// Mitsubishi GX Works2 project: tutor09_webmonitor   PLC: FX1N/FX1NC

PROGRAM MAIN
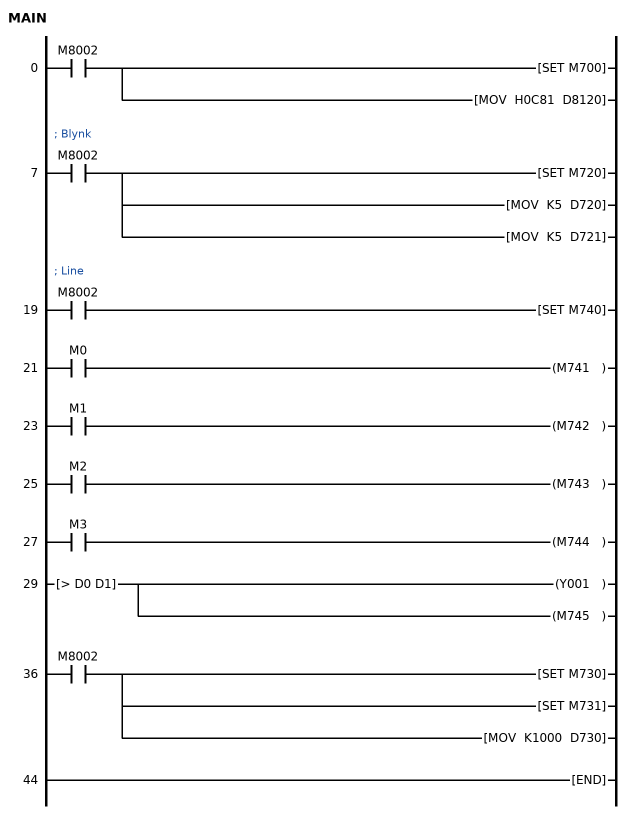
0     LD      M8002
      SET     M700
      MOV     H0C81 D8120
; Blynk
7     LD      M8002
      SET     M720
      MOV     K5 D720
      MOV     K5 D721
; Line
19    LD      M8002
      SET     M740
21    LD      M0
      OUT     M741
23    LD      M1
      OUT     M742
25    LD      M2
      OUT     M743
27    LD      M3
      OUT     M744
29    LD>     D0 D1
      OUT     Y001
      OUT     M745
36    LD      M8002
      SET     M730
      SET     M731
      MOV     K1000 D730
44    END
END_PROGRAM
